// TIA Portal V18 export
// export: Created 2026-06-09T02:47:53.2111236Z, ExportSetting WithDefaults, DisplayName Totally Integrated Automation Portal, DisplayVersion V18, DisplayName TIA Portal Openness, DisplayVersion V18, DisplayName TIA Portal Version Control Interface, DisplayVersion V18, DisplayName STEP 7 Professional, DisplayVersion V18, DisplayName STEP 7 Safety, DisplayVersion V18, DisplayName WinCC Professional, DisplayVersion V18
FUNCTION_BLOCK "Przenosnik tasmowy"   // FB5, LAD
{ S7_Optimized_Access := 'TRUE' }
VERSION : 0.1
// stored: AutoNumber true, IsIECCheckEnabled false, IsRetainMemResEnabled false, MemoryReserve 100, SetENOAutomatically false, UDAEnableTagReadback false
   VAR_TEMP
      mem0 : Time;
   END_VAR
BEGIN

REGION Network 1
   // Start przenośnika taśmowego.
   // Wyłącznik przenośnika znajduje się fizycznie na linii produkcyjnej. Stop natomiast w panelu HMI.
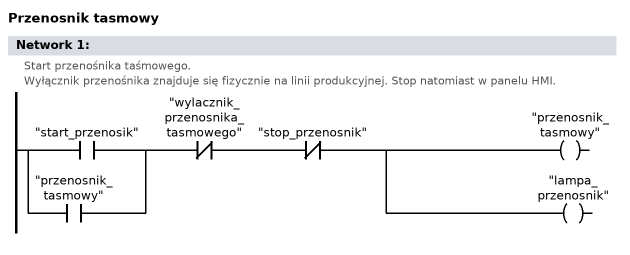
   RUNG wire#powerrail
      Contact( "start_przenosik" )
      wire#w1
      I_Contact( "wylacznik_przenosnika_tasmowego" )
      I_Contact( "stop_przenosnik" )
      wire#w2
      Coil( "przenosnik_tasmowy" )
   END_RUNG
   RUNG wire#powerrail
      Contact( "przenosnik_tasmowy" )
   END_RUNG wire#w1
   RUNG wire#w2
      Coil( "lampa_przenosnik" )
   END_RUNG
   // the same network as SCL:
   "przenosnik_tasmowy" := ("start_przenosik" OR "przenosnik_tasmowy") AND NOT "wylacznik_przenosnika_tasmowego" AND NOT "stop_przenosnik";
   "lampa_przenosnik" := "przenosnik_tasmowy";
END_REGION
END_FUNCTION_BLOCK
